(* CODESYS project tcl_baseclasses.library
   Company: Red Rock Controls Limited
   Description: Naming convention updated
   Version: 1.1.0.0
   Placeholder: tcl_BaseClasses
   Author: Roger Christopher
   Title: tcl_BaseClasses

Project tree, tasks and I/O mapping:
  libraries: Tc2_Standard, * (Beckhoff Automation GmbH); Tc2_System, * (Beckhoff Automation GmbH); Tc2_Utilities, * (Beckhoff Automation GmbH); Tc3_DynamicMemory, * (Beckhoff Automation GmbH); Tc3_EventLogger, * (Beckhoff Automation GmbH); Tc3_Module, * (Beckhoff Automation GmbH); tcl_StringUtils, * (Red Rock Controls Limited)
  Classes/
    Event Framework/
      Event Base Class/
        interface I_Event: AddEventHandler, Args, ClearEventHandlers, Raise
        function block T_EventBase [ST]: AddEventHandler, Args, CallHandler, ClearEventHandlers, IsHandlerSupported, Raise
      Event Handler Base/
        interface I_EventHandlerBase
      List Of Handlers/
        function block T_ListOfEventHandlers [ST]: AddHandler, Clear, Count, FB_exit, FB_init, GetHandler
    Execution/
      Execution/
        interface I_Execution: Abort, Clear, Start, Aborted, Busy, Done, Error, ErrorId, Event_OnAbort, Event_OnError, Notification_OnAbort, Notification_OnError, Ready, Starting
        function block T_Execution [ST]: Abort, Clear, FB_init, SetAborted, SetBusy, SetDone, SetError, Start, Aborted, Aborting, Busy, Done, Error, ErrorId, Event_OnAbort, Event_OnError, Notification_OnAbort, Notification_OnError, Ready, Starting, State
        data type T_ExecutionState
    Function Block Wrappers/
      Classes/
        function block T_Counter [ST]: Dec, Inc, Reset, Value, ValueAsTArg
        function block T_FallingEdge [ST]: EdgeDetected, Test
        function block T_OffTimer [ST]: Delay, FB_init, OutputState, PresetTime
        function block T_OnTimer [ST]: Delay, FB_init, OutputState, PresetTime, Reset, Run
        function block T_PulseTimer [ST]: FB_init, OutputState, PresetTime, Pulse, Reset, Run
        function block T_RisingEdge [ST]: EdgeDetected, Test
        function block T_StructureCrcMonitor [ST]: Changed, Reset, Test
        function block T_ValueMonitor [ST]: Changed, CurrentValue, PreviousValue, Reset, Test
        function block T_ValueMonitorEx [ST]: Changed, Reset, Test
      Event Logging/
        function F_LogError [ST]
        function F_LogMessage [ST]
        function F_LogWarning [ST]
    Notifications/
      Handler Interface/
        interface I_NotificationHandler: OnNotificationReceived
        function block T_NotificationHandler [ST]: IsRaised, NotificationArgs, OnNotificationReceived
      List Of Handlers/
        function block T_ListONotificationHandlers [ST]: AddHandler, Clear, Count, FB_exit, FB_init, GetHandler
      Notification Class/
        interface I_Notification: AddNotificationHandler, ClearNotificationHandlers, Raise, SetNotificationId, Args, Name, NotificationId
        function block T_Notification [ST]: AddNotificationHandler, ClearNotificationHandlers, FB_init, Raise, SetNotificationId, stripName, Args, Name, NotificationId
    Stream/
      interface I_StreamReader: Read_BLOB, Read_BOOL, Read_BYTE, Read_DINT, Read_INT, Read_LINT, Read_LREAL, Read_PVOID, Read_REAL, Read_STRING, Read_UDINT, Read_UINT, Read_ULINT, Seek, BufferAddress, ByteCount, Position, StreamLength
      interface I_StreamWriter: Add_BLOB, Add_BOOL, Add_BYTE, Add_DINT, Add_INT, Add_LINT, Add_LREAL, Add_PVOID, Add_REAL, Add_STRING, Add_UDINT, Add_UINT, Add_ULINT, Clear, Seek
      function block T_Stream [ST]: _ResizeIfNecessary, Add_BLOB, Add_BOOL, Add_BYTE, Add_DINT, Add_INT, Add_LINT, Add_LREAL, Add_PVOID, Add_REAL, Add_STRING, Add_UDINT, Add_UINT, Add_ULINT, Clear, CopyFromStreamReader, FB_exit, FB_init, Init, Read_BLOB, Read_BOOL, Read_BYTE, Read_DINT, Read_INT, Read_LINT, Read_LREAL, Read_PVOID, Read_REAL, Read_STRING, Read_UDINT, Read_UINT, Read_ULINT, Resize, Seek, BufferAddress, ByteCount, Position, StreamLength
  Events/
    Assertion Failed/
      interface I_EventHandler_OnAssertionFailed: OnAssertionFailed
      function block T_Event_AssertionFailed [ST]: CallHandler, IsHandlerSupported
    Execution Aborted/
      interface I_EventHandler_OnExecutionAborted: OnExecutionAborted
      function block T_Event_ExecutionAborted [ST]: CallHandler, IsHandlerSupported
    Execution Failed/
      interface I_EventHandler_OnExecutionFailed: OnExecutionFailed
      function block T_Event_ExecutionFailed [ST]: CallHandler, IsHandlerSupported
  Functions/
    function F_Assert [ST]
    function F_ClearMem [ST]
    function F_DINT_TO_UDINT [ST]
    function F_Equals [ST]
    function F_GetAdsPort [ST]
    function F_GetTaskTime [ST]
    function F_NotEqual [ST]
    function F_UDINT_TO_DINT [ST]
  GVLs/
    global variables GlobalEvents
    global variables GlobalVariables
*)

// Classes/Execution/Execution/T_ExecutionState
{attribute 'qualified_only'}
{attribute 'strict'}
TYPE T_ExecutionState :
(
    Ready := 0,
	Starting,
    Busy,
    Aborting);
END_TYPE

// GVLs/GlobalEvents
(*
Global event instances 
These events are raised by all instances of T_Execution by default when an error occurs
This behaviour can be overidden by setting the Event_OnError or Event_OnAbort properties
of the instance of T_Execution to 0
*)
{attribute 'qualified_only'}
VAR_GLOBAL
    Event_OnError           : T_Event_ExecutionFailed;
    Event_OnAbort           : T_Event_ExecutionAborted;
    Event_AssertionFailed   : T_Event_AssertionFailed;
    
    Notification_ExecutionFailed  : T_Notification;
    Notification_ExecutionAborted : T_Notification;
    Notification_AssertionFailed  : T_Notification;
    
END_VAR

// GVLs/GlobalVariables
{attribute 'qualified_only'}
VAR_GLOBAL
    //Message : FB_TcMessage;
END_VAR

// Classes/Event Framework/Event Base Class/I_Event
INTERFACE I_Event

METHOD AddEventHandler : I_Event
VAR_INPUT
    Handler : I_EventHandlerBase;
END_VAR
END_METHOD

PROPERTY Args : I_StreamWriter
GET
END_GET
END_PROPERTY

METHOD ClearEventHandlers : I_Event
VAR_INPUT
END_VAR
END_METHOD

METHOD Raise
END_METHOD

END_INTERFACE

// Classes/Event Framework/Event Handler Base/I_EventHandlerBase
INTERFACE I_EventHandlerBase EXTENDS __SYSTEM.IQueryInterface

END_INTERFACE

// Classes/Stream/I_StreamWriter
INTERFACE I_StreamWriter

METHOD Add_BLOB : I_StreamWriter
VAR_INPUT
    Value : ANY;
END_VAR
END_METHOD

METHOD Add_BOOL : I_StreamWriter
VAR_INPUT
    Value : BOOL;
END_VAR
END_METHOD

METHOD Add_BYTE : I_StreamWriter
VAR_INPUT
    Value : BYTE;
END_VAR
END_METHOD

METHOD Add_DINT : I_StreamWriter
VAR_INPUT
    Value : DINT;
END_VAR
END_METHOD

METHOD Add_INT : I_StreamWriter
VAR_INPUT
    Value : INT;
END_VAR
END_METHOD

METHOD Add_LINT : I_StreamWriter
VAR_INPUT
    Value : LINT;
END_VAR
END_METHOD

METHOD Add_LREAL : I_StreamWriter
VAR_INPUT
    Value : LREAL;
END_VAR
END_METHOD

METHOD Add_PVOID : I_StreamWriter
VAR_INPUT
    Value : PVOID;
END_VAR
END_METHOD

METHOD Add_REAL : I_StreamWriter
VAR_INPUT
    Value : REAL;
END_VAR
END_METHOD

METHOD Add_STRING : I_StreamWriter
VAR_INPUT
    Value : STRING(255);
END_VAR
END_METHOD

METHOD Add_UDINT : I_StreamWriter
VAR_INPUT
    Value : UDINT;
END_VAR
END_METHOD

METHOD Add_UINT : I_StreamWriter
VAR_INPUT
    Value : UINT;
END_VAR
END_METHOD

METHOD Add_ULINT : I_StreamWriter
VAR_INPUT
    Value : ULINT;
END_VAR
END_METHOD

METHOD Clear : I_StreamWriter
END_METHOD

METHOD Seek: I_StreamWriter
VAR_INPUT
    Position : UDINT;
END_VAR
END_METHOD

END_INTERFACE

// Classes/Event Framework/Event Base Class/T_EventBase
{attribute 'reflection'}
FUNCTION_BLOCK ABSTRACT T_EventBase IMPLEMENTS I_Event
VAR
    EventHandlers : T_ListOfEventHandlers(Capacity := 5);
    
    {attribute 'instance-path'} {attribute 'no_init'}
    EventName : T_MaxString; // Automatically initialised with the full name of the instance   
    
    EventArgs : T_Stream(StreamLength := 8);
    
    Message_EventHandlerNotImplemented : FB_TcMessage;
END_VAR

METHOD AddEventHandler : I_Event
VAR_INPUT
    Handler : I_EventHandlerBase;
END_VAR
IF IsHandlerSupported(Handler) THEN
    EventHandlers.AddHandler(Handler);
//ELSE
//    IF Message_EventHandlerNotImplemented.nEventId = 0 THEN
//        Message_EventHandlerNotImplemented.CreateEx(
//            stEventEntry := TC_EVENTS.tcl_BaseClassEvents.EventHandlerNotImplemented,
//            ipSourceInfo := 0);
//    END_IF
//    Message_EventHandlerNotImplemented.Send(0);

END_IF
AddEventHandler := THIS^;
END_METHOD

PROPERTY PUBLIC Args : I_StreamWriter
GET
Args := EventArgs;
END_GET
END_PROPERTY

METHOD ABSTRACT CallHandler
VAR_INPUT
    HandlerBase : I_EventHandlerBase;
    EventArgs : I_StreamReader;
END_VAR
END_METHOD

METHOD ClearEventHandlers : I_Event
EventHandlers.Clear();
ClearEventHandlers := THIS^;
END_METHOD

METHOD ABSTRACT IsHandlerSupported : BOOL
VAR_INPUT
    HandlerBase : I_EventHandlerBase;
END_VAR
END_METHOD

METHOD Raise
VAR
    HandlerBase : I_EventHandlerBase;
    i : UDINT;
END_VAR
IF EventHandlers.Count > 0 THEN
    FOR i := 0 TO EventHandlers.Count - 1 DO
        HandlerBase := EventHandlers.GetHandler(i);
        IF HandlerBase <> 0 THEN
            EventArgs.Seek(0); // to ensure that each handler reads args from start of the stream
            CallHandler(HandlerBase,EventArgs);
        END_IF
    END_FOR
END_IF
EventArgs.Clear(); // to leave event args empty for next time event is raised
END_METHOD

END_FUNCTION_BLOCK

// Classes/Event Framework/List Of Handlers/T_ListOfEventHandlers
{attribute 'hide'}
FUNCTION_BLOCK T_ListOfEventHandlers
VAR
    Buffer : FB_DynMem_Buffer(ipMemMan:= DynamicMemoryManager);
    DynamicMemoryManager : FB_DynMem_Manager;

    pHandler : POINTER TO I_EventHandlerBase;
    HandlerCount : UDINT;
    Capacity : UDINT;
END_VAR

METHOD AddHandler
VAR_INPUT
    Handler : I_EventHandlerBase;
END_VAR
IF Count = Capacity THEN
    Capacity := Capacity * 2;
    Buffer.Resize(
        nSize     := Capacity * SIZEOF(PVOID),
        bPreserve := TRUE,
        bReset    := FALSE);
    pHandler := Buffer.pBuffer;
END_IF

pHandler[HandlerCount] := Handler;
HandlerCount := HandlerCount + 1;
END_METHOD

METHOD Clear
VAR_INPUT
END_VAR
Buffer.Clear();
HandlerCount := 0;
END_METHOD

PROPERTY Count : UDINT
GET
Count := HandlerCount;
END_GET
END_PROPERTY

METHOD FB_exit : BOOL
VAR_INPUT
	bInCopyCode : BOOL; // if TRUE, the exit method is called for exiting an instance that is copied afterwards (online change).
END_VAR
IF NOT bInCopyCode THEN
    Buffer.DeleteBuffer();
    pHandler := 0;
END_IF
END_METHOD

METHOD FB_init : BOOL
VAR_INPUT
	bInitRetains : BOOL; // if TRUE, the retain variables are initialized (warm start / cold start)
	bInCopyCode : BOOL;  // if TRUE, the instance afterwards gets moved into the copy code (online change)
    Capacity : UDINT;
END_VAR
Buffer.CreateBuffer(
    nSize := Capacity * SIZEOF(PVOID),
    bReset := TRUE);
    
pHandler := Buffer.pBuffer;
THIS^.Capacity := Capacity;
END_METHOD

METHOD GetHandler : I_EventHandlerBase
VAR_INPUT
    Index : UDINT;
END_VAR
IF Index < HandlerCount AND Index >= 0 THEN 
    GetHandler := pHandler[Index];
END_IF
END_METHOD

END_FUNCTION_BLOCK

// Classes/Stream/T_Stream
FUNCTION_BLOCK T_Stream IMPLEMENTS I_StreamWriter, I_StreamReader
VAR
    
    MemoryManager : FB_DynMem_Manager;
    Buffer : FB_DynMem_Buffer(ipMemMan:= MemoryManager);
    pBuffer : POINTER TO BYTE;
    
    _StreamLength : UDINT := 4;
    _Position : UDINT;
    _ByteCount : UDINT;
END_VAR

METHOD PRIVATE _ResizeIfNecessary
VAR_INPUT
    SpaceRequired : UDINT;
END_VAR
IF _Position + SpaceRequired > _StreamLength THEN
    Resize(StreamLength := _Position + SpaceRequired);
END_IF
END_METHOD

METHOD Add_BLOB : I_StreamWriter
VAR_INPUT
    Value : ANY;
END_VAR
VAR
    pValue : POINTER TO BYTE;
END_VAR
_ResizeIfNecessary(SpaceRequired := DINT_TO_UDINT(Value.diSize));

MEMCPY(
    destAddr:= pBuffer + _Position, 
    srcAddr := Value.pValue, 
    n       := DINT_TO_UDINT(Value.diSize));

_Position  := _Position + DINT_TO_UDINT(Value.diSize); 
_ByteCount := _ByteCount + DINT_TO_UDINT(Value.diSize); 
   
Add_BLOB := THIS^;
END_METHOD

METHOD Add_BOOL : I_StreamWriter
VAR_INPUT
    Value : BOOL;
END_VAR
VAR
    pValue : POINTER TO BOOL;
END_VAR
_ResizeIfNecessary(SpaceRequired := SIZEOF(Value));

pValue := pBuffer + _Position;
pValue^ := Value;
_Position := _Position + SIZEOF(Value); 
_ByteCount := _ByteCount + SIZEOF(Value); 
   
Add_BOOL := THIS^;
END_METHOD

METHOD Add_BYTE : I_StreamWriter
VAR_INPUT
    Value : BYTE;
END_VAR
VAR
    pValue : POINTER TO BYTE;
END_VAR
_ResizeIfNecessary(SpaceRequired := SIZEOF(Value));

pValue := pBuffer + _Position;
pValue^ := Value;
_Position := _Position + SIZEOF(Value); 
_ByteCount := _ByteCount + SIZEOF(Value); 

Add_BYTE := THIS^;
END_METHOD

METHOD Add_DINT : I_StreamWriter
VAR_INPUT
    Value : DINT;
END_VAR
VAR
    pValue : POINTER TO DINT;
END_VAR
_ResizeIfNecessary(SpaceRequired := SIZEOF(Value));

pValue := pBuffer + _Position;
pValue^ := Value;
_Position := _Position + SIZEOF(Value); 
_ByteCount := _ByteCount + SIZEOF(Value); 

   
Add_DINT := THIS^;
END_METHOD

METHOD Add_INT : I_StreamWriter
VAR_INPUT
    Value : INT;
END_VAR
VAR
    pValue : POINTER TO INT;
END_VAR
_ResizeIfNecessary(SpaceRequired := SIZEOF(Value));

pValue := pBuffer + _Position;
pValue^ := Value;
_Position := _Position + SIZEOF(Value);    
_ByteCount := _ByteCount + SIZEOF(Value); 


Add_INT := THIS^;
END_METHOD

METHOD Add_LINT : I_StreamWriter
VAR_INPUT
    Value : LINT;
END_VAR
VAR
    pValue : POINTER TO LINT;
END_VAR
_ResizeIfNecessary(SpaceRequired := SIZEOF(Value));

pValue := pBuffer + _Position;
pValue^ := Value;
_Position := _Position + SIZEOF(Value); 
_ByteCount := _ByteCount + SIZEOF(Value); 

   
Add_LINT := THIS^;
END_METHOD

METHOD Add_LREAL : I_StreamWriter
VAR_INPUT
    Value : LREAL;
END_VAR
VAR
    pValue : POINTER TO LREAL;
END_VAR
_ResizeIfNecessary(SpaceRequired := SIZEOF(Value));

pValue := pBuffer + _Position;
pValue^ := Value;
_Position := _Position + SIZEOF(Value);    
_ByteCount := _ByteCount + SIZEOF(Value); 


Add_LREAL := THIS^;
END_METHOD

METHOD Add_PVOID : I_StreamWriter
VAR_INPUT
    Value : PVOID;
END_VAR
VAR
    pValue : POINTER TO PVOID;
END_VAR
_ResizeIfNecessary(SpaceRequired := SIZEOF(Value));

pValue := pBuffer + _Position;
pValue^ := Value;
_Position := _Position + SIZEOF(Value); 
_ByteCount := _ByteCount + SIZEOF(Value); 

   
Add_PVOID := THIS^;
END_METHOD

METHOD Add_REAL : I_StreamWriter
VAR_INPUT
    Value : REAL;
END_VAR
VAR
    pValue : POINTER TO REAL;
END_VAR
_ResizeIfNecessary(SpaceRequired := SIZEOF(Value));

pValue := pBuffer + _Position;
pValue^ := Value;
_Position := _Position + SIZEOF(Value);    
_ByteCount := _ByteCount + SIZEOF(Value); 


Add_REAL := THIS^;
END_METHOD

METHOD Add_STRING : I_StreamWriter // adds any string length as we only store the chars + null byte
VAR_INPUT
    Value : STRING(255);
END_VAR
VAR
    StringSize : UDINT; // number of characters plus the null termination byte
END_VAR
StringSize := INT_TO_UDINT(LEN(Value) + 1);

_ResizeIfNecessary(SpaceRequired := StringSize);  // only storing the characters and the null termination byte

MEMCPY(
    destAddr := pBuffer + _Position,
    srcAddr  := ADR(Value),
    n        := StringSize);


_Position := _Position + StringSize;    
_ByteCount := _ByteCount + StringSize; 


Add_STRING := THIS^;
END_METHOD

METHOD Add_UDINT : I_StreamWriter
VAR_INPUT
    Value : UDINT;
END_VAR
VAR
    pValue : POINTER TO UDINT;
END_VAR
_ResizeIfNecessary(SpaceRequired := SIZEOF(Value));

pValue := pBuffer + _Position;
pValue^ := Value;
_Position := _Position + SIZEOF(Value);    
_ByteCount := _ByteCount + SIZEOF(Value); 


Add_UDINT := THIS^;
END_METHOD

METHOD Add_UINT : I_StreamWriter
VAR_INPUT
    Value : UINT;
END_VAR
VAR
    pValue : POINTER TO UINT;
END_VAR
_ResizeIfNecessary(SpaceRequired := SIZEOF(Value));

pValue := pBuffer + _Position;
pValue^ := Value;
_Position := _Position + SIZEOF(Value);    
_ByteCount := _ByteCount + SIZEOF(Value); 


Add_UINT := THIS^;
END_METHOD

METHOD Add_ULINT : I_StreamWriter
VAR_INPUT
    Value : ULINT;
END_VAR
VAR
    pValue : POINTER TO ULINT;
END_VAR
_ResizeIfNecessary(SpaceRequired := SIZEOF(Value));

pValue := pBuffer + _Position;
pValue^ := Value;
_Position := _Position + SIZEOF(Value); 
_ByteCount := _ByteCount + SIZEOF(Value); 

   
Add_ULINT := THIS^;
END_METHOD

METHOD Clear : I_StreamWriter
Buffer.Clear();
_Position := 0;
_ByteCount := 0;
pBuffer := Buffer.pBuffer;
Clear := THIS^;
END_METHOD

METHOD CopyFromStreamReader
VAR_INPUT
    StreamToCopyFrom : I_StreamReader;
END_VAR
IF StreamToCopyFrom.StreamLength > THIS^.StreamLength THEN
    Resize(StreamToCopyFrom.StreamLength);
END_IF

MEMCPY(
    destAddr := Buffer.pBuffer,
    srcAddr  := StreamToCopyFrom.BufferAddress,
    n        := StreamToCopyFrom.StreamLength);
    
THIS^._ByteCount    := StreamToCopyFrom.ByteCount;
THIS^._StreamLength := StreamToCopyFrom.StreamLength;
THIS^._Position     := 0;
END_METHOD

METHOD FB_exit : BOOL
VAR_INPUT
	bInCopyCode : BOOL; // if TRUE, the exit method is called for exiting an instance that is copied afterwards (online change).
END_VAR
IF NOT bInCopyCode THEN
    Buffer.DeleteBuffer();
END_IF
END_METHOD

METHOD FB_init : BOOL
VAR_INPUT
	bInitRetains : BOOL; // if TRUE, the retain variables are initialized (warm start / cold start)
	bInCopyCode : BOOL;  // if TRUE, the instance afterwards gets moved into the copy code (online change)
    StreamLength : UDINT;
END_VAR
IF NOT bInCopyCode THEN
    Init(StreamLength);
END_IF
END_METHOD

METHOD Init
VAR_INPUT
    StreamLength : UDINT;
END_VAR
IF Buffer.bAvailable THEN
    Buffer.DeleteBuffer();
END_IF

_StreamLength := StreamLength;
Buffer.CreateBuffer(nSize := _StreamLength, bReset := TRUE);
_Position := 0;
_ByteCount := 0;
pBuffer := Buffer.pBuffer;
END_METHOD

METHOD Read_BLOB
VAR_INPUT
    Value : ANY;
END_VAR

VAR
    pValue : POINTER TO BYTE;
    Result : BYTE;
END_VAR
IF _Position + DINT_TO_UDINT(Value.diSize) <= _StreamLength THEN
    
MEMCPY(
    destAddr:= Value.pValue, 
    srcAddr := pBuffer + _Position, 
    n       := DINT_TO_UDINT(Value.diSize));

    _Position := _Position + DINT_TO_UDINT(Value.diSize);   
END_IF
END_METHOD

METHOD Read_BOOL : BOOL;
VAR
    pValue : POINTER TO BOOL;
    Result : BOOL;
END_VAR
IF _Position + SIZEOF(Result) <= _StreamLength THEN
    pValue := pBuffer + _Position;
    Result := pValue^;
    _Position := _Position + SIZEOF(Result);   
    Read_BOOL := Result; 
END_IF
END_METHOD

METHOD Read_BYTE : BYTE;
VAR
    pValue : POINTER TO BYTE;
    Result : BYTE;
END_VAR
IF _Position + SIZEOF(Result) <= _StreamLength THEN
    pValue := pBuffer + _Position;
    Result := pValue^;
    _Position := _Position + SIZEOF(Result);   
    Read_BYTE := Result; 
END_IF
END_METHOD

METHOD Read_DINT : DINT;
VAR
    pValue : POINTER TO DINT;
    Result : DINT;
END_VAR
IF _Position + SIZEOF(Result) <= _StreamLength THEN
    pValue := pBuffer + _Position;
    Result := pValue^;
    _Position := _Position + SIZEOF(Result);   
    Read_DINT := Result; 
END_IF
END_METHOD

METHOD Read_INT : INT;
VAR
    pValue : POINTER TO INT;
    Result : INT;
END_VAR
IF _Position + SIZEOF(Result) <= _StreamLength THEN
    pValue := pBuffer + _Position;
    Result := pValue^;
    _Position := _Position + SIZEOF(Result);   
    Read_INT := Result; 
END_IF
END_METHOD

METHOD Read_LINT : LINT;
VAR
    pValue : POINTER TO LINT;
    Result : LINT;
END_VAR
IF _Position + SIZEOF(Result) <= _StreamLength THEN
    pValue := pBuffer + _Position;
    Result := pValue^;
    _Position := _Position + SIZEOF(Result);   
    Read_LINT := Result; 
END_IF
END_METHOD

METHOD Read_LREAL : LREAL;
VAR
    pValue : POINTER TO LREAL;
    Result : LREAL;
END_VAR
IF _Position + SIZEOF(Result) <= _StreamLength THEN
    pValue := pBuffer + _Position;
    Result := pValue^;
    _Position := _Position + SIZEOF(Result);   
    Read_LREAL := Result; 
END_IF
END_METHOD

METHOD Read_PVOID : PVOID;
VAR
    pValue : POINTER TO PVOID;
    Result : PVOID;
END_VAR
IF _Position + SIZEOF(Result) <= _StreamLength THEN
    pValue := pBuffer + _Position;
    Result := pValue^;
    _Position := _Position + SIZEOF(Result);   
    Read_PVOID := Result; 
END_IF
END_METHOD

METHOD Read_REAL : REAL;
VAR
    pValue : POINTER TO REAL;
    Result : REAL;
END_VAR
IF _Position + SIZEOF(Result) <= _StreamLength THEN
    pValue := pBuffer + _Position;
    Result := pValue^;
    _Position := _Position + SIZEOF(Result);   
    Read_REAL := Result; 
END_IF
END_METHOD

METHOD Read_STRING : STRING(255);
VAR
    pValue : POINTER TO STRING(255);
    StringSize : UDINT; // number of characters plus the null termination byte
END_VAR
pValue := pBuffer + _Position;

StringSize := INT_TO_UDINT(LEN(pValue^) + 1);

IF _Position + StringSize <= _StreamLength THEN // end of string is in the buffer, so proceed...
    _Position := _Position + StringSize;   
    Read_STRING := pValue^;
END_IF
END_METHOD

METHOD Read_UDINT : UDINT;
VAR
    pValue : POINTER TO UDINT;
    Result : UDINT;
END_VAR
IF _Position + SIZEOF(Result) <= _StreamLength THEN
    pValue := pBuffer + _Position;
    Result := pValue^;
    _Position := _Position + SIZEOF(Result);   
    Read_UDINT := Result; 
END_IF
END_METHOD

METHOD Read_UINT : UINT;
VAR
    pValue : POINTER TO UINT;
    Result : UINT;
END_VAR
IF _Position + SIZEOF(Result) <= _StreamLength THEN
    pValue := pBuffer + _Position;
    Result := pValue^;
    _Position := _Position + SIZEOF(Result);   
    Read_UINT := Result; 
END_IF
END_METHOD

METHOD Read_ULINT : ULINT;
VAR
    pValue : POINTER TO ULINT;
    Result : ULINT;
END_VAR
IF _Position + SIZEOF(Result) <= _StreamLength THEN
    pValue := pBuffer + _Position;
    Result := pValue^;
    _Position := _Position + SIZEOF(Result);   
    Read_ULINT := Result; 
END_IF
END_METHOD

METHOD Resize
VAR_INPUT
    StreamLength : UDINT;
END_VAR
Buffer.Resize(nSize := StreamLength, bPreserve := TRUE, bReset := FALSE);
_StreamLength := StreamLength;
pBuffer := Buffer.pBuffer;
END_METHOD

METHOD Seek : I_StreamWriter
VAR_INPUT
    Position : UDINT;
END_VAR
IF Position <= _StreamLength THEN
    THIS^._Position := Position;
END_IF
Seek := THIS^;
END_METHOD

PROPERTY BufferAddress : PVOID
GET
BufferAddress := Buffer.pBuffer;
END_GET
END_PROPERTY

PROPERTY ByteCount : UDINT
GET
ByteCount := _ByteCount;
END_GET
END_PROPERTY

PROPERTY Position : UDINT
GET
Position := _Position;
END_GET
END_PROPERTY

PROPERTY StreamLength : UDINT
GET
StreamLength := _StreamLength;
END_GET
END_PROPERTY

END_FUNCTION_BLOCK

// Classes/Stream/I_StreamReader
INTERFACE I_StreamReader

METHOD Read_BLOB
VAR_INPUT
    Value : ANY;
END_VAR
END_METHOD

METHOD Read_BOOL : BOOL;
END_METHOD

METHOD Read_BYTE : BYTE;
END_METHOD

METHOD Read_DINT : DINT;
END_METHOD

METHOD Read_INT : INT;
END_METHOD

METHOD Read_LINT : LINT;
END_METHOD

METHOD Read_LREAL : LREAL;
END_METHOD

METHOD Read_PVOID : PVOID;
END_METHOD

METHOD Read_REAL : REAL;
END_METHOD

METHOD Read_STRING : STRING(255);
END_METHOD

METHOD Read_UDINT : UDINT;
END_METHOD

METHOD Read_UINT : UINT;
END_METHOD

METHOD Read_ULINT : ULINT;
END_METHOD

METHOD Seek: I_StreamWriter
VAR_INPUT
    Position : UDINT;
END_VAR
END_METHOD

PROPERTY BufferAddress : PVOID
GET
END_GET
END_PROPERTY

PROPERTY ByteCount : UDINT
GET
END_GET
END_PROPERTY

PROPERTY Position : UDINT
GET
END_GET
END_PROPERTY

PROPERTY StreamLength : UDINT
GET
END_GET
END_PROPERTY

END_INTERFACE

// Classes/Execution/Execution/I_Execution
INTERFACE I_Execution

METHOD Abort 
VAR_INPUT
END_VAR
END_METHOD

METHOD Clear 
VAR_INPUT
END_VAR
END_METHOD

METHOD Start : BOOL // returns TRUE if start request accepted (i.e State was Ready)
VAR_INPUT
END_VAR
END_METHOD

PROPERTY Aborted : BOOL
GET
END_GET
END_PROPERTY

PROPERTY Busy : BOOL
GET
END_GET
END_PROPERTY

PROPERTY Done : BOOL
GET
END_GET
END_PROPERTY

PROPERTY Error : BOOL
GET
END_GET
END_PROPERTY

PROPERTY ErrorId : UDINT
GET
END_GET
END_PROPERTY

PROPERTY Event_OnAbort : I_Event
GET
END_GET
SET
END_SET
END_PROPERTY

PROPERTY Event_OnError : I_Event
GET
END_GET
SET
END_SET
END_PROPERTY

PROPERTY Notification_OnAbort : I_Notification
GET
END_GET
SET
END_SET
END_PROPERTY

PROPERTY Notification_OnError : I_Notification
GET
END_GET
SET
END_SET
END_PROPERTY

PROPERTY Ready : BOOL
GET
END_GET
END_PROPERTY

PROPERTY Starting : BOOL
GET
END_GET
END_PROPERTY

END_INTERFACE

// Classes/Notifications/Notification Class/I_Notification
INTERFACE I_Notification

METHOD AddNotificationHandler : I_Notification
VAR_INPUT
    Handler : I_NotificationHandler;
END_VAR
END_METHOD

METHOD ClearNotificationHandlers : I_Notification
VAR_INPUT
END_VAR
END_METHOD

METHOD Raise
END_METHOD

METHOD SetNotificationId : I_Notification
VAR_INPUT
    NotificationId : UDINT;
END_VAR
END_METHOD

PROPERTY Args : I_StreamWriter
GET
END_GET
END_PROPERTY

PROPERTY Name : T_MaxString
GET
END_GET
END_PROPERTY

PROPERTY NotificationId : UDINT
GET
END_GET
SET
END_SET
END_PROPERTY

END_INTERFACE

// Classes/Notifications/Handler Interface/I_NotificationHandler
INTERFACE I_NotificationHandler EXTENDS __SYSTEM.IQueryInterface

METHOD OnNotificationReceived
VAR_INPUT
    NotificationId   : UDINT;
    NotificationName : T_MaxString;
    Args             : I_StreamReader;
END_VAR
END_METHOD

END_INTERFACE

// Classes/Execution/Execution/T_Execution
(*
:Class for handling communications between a client requesting a service 
:and a server providing the service
*)
{attribute 'reflection'}
FUNCTION_BLOCK T_Execution IMPLEMENTS I_Execution
VAR
    _State      : T_ExecutionState;
    _Done       : BOOL;
    _Error      : BOOL;
    _Aborted    : BOOL;
    
    {attribute 'displaymode':='hex'}
    _ErrorId    : UDINT;
    
    {attribute 'instance-path'} {attribute 'no_init'}
    Name        : T_MaxString; // Automatically initialised with the full name of the instance
    
    _Event_OnError : I_Event;
    _Event_OnAbort : I_Event;
    
    _Notification_OnError : I_Notification;
    _Notification_OnAbort : I_Notification;
    
    SourceInfo : FB_TcSourceInfo;
    
    Message_ExecutionError : FB_TcMessage;
    Message_ExecutionAborted : FB_TcMessage;
    Message_ExecutionNotReady : FB_TcMessage;
END_VAR

// Requests that the current operation be aborted - set the State to Aborting
METHOD Abort
// Aborting must be handled by parent class - cleanup and set Ready state
_State := T_ExecutionState.Aborting;
END_METHOD

// Clears the results flags provided State = Ready
METHOD Clear
IF _State = T_ExecutionState.Ready  THEN
    _Done    := FALSE;
    _Aborted := FALSE;
    _Error   := FALSE;
    _ErrorId := 0;
    
ELSE
    IF _Event_OnError <> 0 THEN
        _Event_OnError.Args.Add_STRING(F_FormatString1(
                                        Format := 'Clear requested while not ready in %s',
                                        Arg1   := F_STRING(Name)));
        _Event_OnError.Raise();
    END_IF
END_IF
END_METHOD

// Individual T_Execution events are assigned here to the global events 
// so by default, all errors/aborts raise these global events
// This can be overidden for individual instances or T_Execution 
// by setting the Event properties to zero (or another event)
METHOD FB_init : BOOL
VAR_INPUT
	bInitRetains : BOOL; // if TRUE, the retain variables are initialized (warm start / cold start)
	bInCopyCode : BOOL;  // if TRUE, the instance afterwards gets moved into the copy code (online change)
END_VAR
_Event_OnAbort := GlobalEvents.Event_OnAbort;
_Event_OnError := GlobalEvents.Event_OnError;
_Notification_OnAbort := GlobalEvents.Notification_ExecutionAborted;
_Notification_OnError := GlobalEvents.Notification_ExecutionFailed;

SourceInfo.sName := Name;
END_METHOD

METHOD SetAborted // used when implementing class signals Aborted
VAR
    EventData : T_MaxString;
END_VAR
IF _State = T_ExecutionState.Starting OR _State = T_ExecutionState.Busy THEN
    _Aborted := TRUE;
    _State := T_ExecutionState.Ready;
    
    IF _Event_OnAbort <> 0 THEN
        _Event_OnAbort.Args.Add_STRING(F_FormatString1('Execution aborted in %s',F_STRING(Name)));
        _Event_OnAbort.Raise();
    END_IF  

    IF _Notification_OnAbort <> 0 THEN
        _Notification_OnAbort.Args.Add_STRING(F_FormatString1('Execution aborted in %s',F_STRING(Name)));
        _Notification_OnAbort.Raise();
    END_IF  

//    IF Message_ExecutionAborted.nEventId = 0 THEN
//        Message_ExecutionAborted.CreateEx(
//            stEventEntry := TC_EVENTS.tcl_BaseClassEvents.ExecutionAborted,
//            ipSourceInfo := 0);
//    END_IF
//    Message_ExecutionAborted.Send(0);
END_IF

IF _State = T_ExecutionState.Aborting THEN
    _Aborted := TRUE;
    _State := T_ExecutionState.Ready;
END_IF
END_METHOD

METHOD SetBusy
VAR_INPUT
END_VAR
IF _State = T_ExecutionState.Starting THEN
    _State := T_ExecutionState.Busy;
END_IF
END_METHOD

METHOD SetDone
VAR_INPUT
END_VAR
IF _State = T_ExecutionState.Starting OR _State = T_ExecutionState.Busy THEN
    _Done := TRUE;
    _State := T_ExecutionState.Ready;
END_IF
END_METHOD

METHOD SetError
VAR_INPUT
    ErrorId : UDINT;
END_VAR
IF _State = T_ExecutionState.Starting OR _State = T_ExecutionState.Busy THEN
    _Error   := TRUE;
    _ErrorId := ErrorId;
    _State   := T_ExecutionState.Ready;
    
    IF _Event_OnError <> 0 THEN
        _Event_OnError.Args.Add_STRING(F_FormatString2('Error 0x%0.4X in %s',F_UDINT(_ErrorId),F_STRING(Name)));
        _Event_OnError.Raise();
    END_IF
    
    IF _Notification_OnError <> 0 THEN
        _Notification_OnError.Args.Add_STRING(F_FormatString2('Error 0x%0.4X in %s',F_UDINT(_ErrorId),F_STRING(Name)));
        _Notification_OnError.Raise();
    END_IF
    
//    IF Message_ExecutionError.nEventId = 0 THEN
//        Message_ExecutionError.CreateEx(
//            stEventEntry := TC_EVENTS.tcl_BaseClassEvents.ExecutionError,
//            ipSourceInfo := 0);
//	END_IF
//    Message_ExecutionError.ipArguments.Clear().AddUDInt(_ErrorId);
//    Message_ExecutionError.Send(0);
END_IF
END_METHOD

METHOD Start : BOOL
VAR_INPUT
END_VAR
IF _State = T_ExecutionState.Ready  THEN
    _Done    := FALSE;
    _Aborted := FALSE;
    _Error   := FALSE;
    _ErrorId := 0;
    
    _State   := T_ExecutionState.Starting;
    Start    := TRUE; // Accepted
ELSE
    IF _Event_OnError <> 0 THEN
        _Event_OnError.Args.Add_STRING(F_FormatString1(
                                        Format := 'Start requested while not ready in %s',
                                        Arg1   := F_STRING(Name)));
        _Event_OnError.Raise();
    END_IF
    
//    IF Message_ExecutionNotReady.nEventId = 0 THEN
//        Message_ExecutionNotReady.CreateEx(
//            stEventEntry := TC_EVENTS.tcl_BaseClassEvents.ExecutionNotReady,
//            ipSourceInfo := 0);
//    END_IF
//    Message_ExecutionNotReady.Send(0);
    
END_IF
END_METHOD

PROPERTY Aborted : BOOL
GET
Aborted := _Aborted;
END_GET
END_PROPERTY

PROPERTY Aborting : BOOL
GET
Aborting := _State = T_ExecutionState.Aborting;
END_GET
END_PROPERTY

PROPERTY Busy : BOOL
GET
Busy := _State = T_ExecutionState.Busy;
END_GET
END_PROPERTY

PROPERTY Done : BOOL
GET
Done := _Done;
END_GET
END_PROPERTY

PROPERTY Error : BOOL
GET
Error := _Error;
END_GET
END_PROPERTY

PROPERTY ErrorId : UDINT
GET
ErrorId := _ErrorId;
END_GET
SET
_ErrorId := ErrorId;
END_SET
END_PROPERTY

PROPERTY Event_OnAbort : I_Event
GET
Event_OnAbort := _Event_OnAbort;
END_GET
SET
_Event_OnAbort := Event_OnAbort;
END_SET
END_PROPERTY

PROPERTY Event_OnError : I_Event
GET
Event_OnError := _Event_OnError;
END_GET
SET
_Event_OnError := Event_OnError;
END_SET
END_PROPERTY

PROPERTY Notification_OnAbort : I_Notification
GET
Notification_OnAbort := _Notification_OnAbort;
END_GET
SET
_Notification_OnAbort := Notification_OnAbort;
END_SET
END_PROPERTY

PROPERTY Notification_OnError : I_Notification
GET
Notification_OnError := _Notification_OnError;
END_GET
SET
_Notification_OnError := Notification_OnError;
END_SET
END_PROPERTY

PROPERTY Ready : BOOL
GET
Ready := _State = T_ExecutionState.Ready;
END_GET
END_PROPERTY

PROPERTY Starting : BOOL
GET
Starting := _State = T_ExecutionState.Starting;
END_GET
END_PROPERTY

PROPERTY State : T_ExecutionState
GET
State := _State;
END_GET
END_PROPERTY

END_FUNCTION_BLOCK

// Classes/Function Block Wrappers/Classes/T_Counter
FUNCTION_BLOCK T_Counter
VAR
    Count : DINT;
END_VAR

METHOD Dec : DINT
VAR_INPUT
END_VAR
Count := Count - 1;
Dec := Count;
END_METHOD

METHOD Inc : DINT
VAR_INPUT
END_VAR
Count := Count + 1;
Inc := Count;
END_METHOD

METHOD Reset
VAR_INPUT
END_VAR
Count := 0;
END_METHOD

PROPERTY Value : DINT
GET
Value := Count;
END_GET
SET
Count := Value;
END_SET
END_PROPERTY

PROPERTY ValueAsTArg : T_Arg
GET
ValueAsTArg := F_DINT(Count);
END_GET
END_PROPERTY

END_FUNCTION_BLOCK

// Classes/Function Block Wrappers/Classes/T_FallingEdge
FUNCTION_BLOCK T_FallingEdge
VAR
    F_TRIG1 : F_TRIG;
END_VAR

PROPERTY EdgeDetected : BOOL
GET
EdgeDetected := F_TRIG1.Q;
END_GET
END_PROPERTY

METHOD Test : BOOL
VAR_INPUT
    Value : BOOL;
END_VAR
F_TRIG1(CLK := Value);
Test := F_TRIG1.Q;
END_METHOD

END_FUNCTION_BLOCK

// Classes/Function Block Wrappers/Classes/T_OffTimer
FUNCTION_BLOCK T_OffTimer
VAR
    TOF1 : TOF;
END_VAR

METHOD Delay : BOOL
VAR_INPUT
    In : BOOL;
END_VAR
TOF1(IN := In);
Delay := TOF1.Q;
END_METHOD

METHOD FB_init : BOOL
VAR_INPUT
	bInitRetains : BOOL; // if TRUE, the retain variables are initialized (warm start / cold start)
	bInCopyCode : BOOL;  // if TRUE, the instance afterwards gets moved into the copy code (online change)
    PresetTime : LREAL; // seconds
END_VAR
TOF1.PT := LREAL_TO_TIME(PresetTime * 1000);
END_METHOD

PROPERTY OutputState : BOOL
GET
OutputState := TOF1.Q;
END_GET
END_PROPERTY

PROPERTY PresetTime : LREAL
GET
PresetTime := TIME_TO_LREAL(TOF1.PT)/1000.0; // in seconds
END_GET
SET
TOF1.PT := LREAL_TO_TIME(PresetTime * 1000);
END_SET
END_PROPERTY

END_FUNCTION_BLOCK

// Classes/Function Block Wrappers/Classes/T_OnTimer
FUNCTION_BLOCK T_OnTimer
VAR
    TON1 : TON;
END_VAR

METHOD Delay : BOOL
VAR_INPUT
    In : BOOL;
END_VAR
TON1(IN := In);
Delay := TON1.Q;
END_METHOD

METHOD FB_init : BOOL
VAR_INPUT
	bInitRetains : BOOL; // if TRUE, the retain variables are initialized (warm start / cold start)
	bInCopyCode : BOOL;  // if TRUE, the instance afterwards gets moved into the copy code (online change)
    PresetTime : LREAL; // seconds
END_VAR
TON1.PT := LREAL_TO_TIME(PresetTime * 1000);
END_METHOD

PROPERTY OutputState : BOOL
GET
OutputState := TON1.Q;
END_GET
END_PROPERTY

PROPERTY PresetTime : LREAL
GET
PresetTime := TIME_TO_LREAL(TON1.PT)/1000.0; // in seconds
END_GET
SET
TON1.PT := LREAL_TO_TIME(PresetTime * 1000);
END_SET
END_PROPERTY

METHOD Reset
TON1(IN := FALSE);
END_METHOD

METHOD Run : BOOL
TON1(IN := TRUE);
Run := TON1.Q;
END_METHOD

END_FUNCTION_BLOCK

// Classes/Function Block Wrappers/Classes/T_PulseTimer
FUNCTION_BLOCK T_PulseTimer
VAR
    TP1 : TP;
END_VAR

METHOD FB_init : BOOL
VAR_INPUT
	bInitRetains : BOOL; // if TRUE, the retain variables are initialized (warm start / cold start)
	bInCopyCode : BOOL;  // if TRUE, the instance afterwards gets moved into the copy code (online change)
    PresetTime : LREAL; // seconds
END_VAR
TP1.PT := LREAL_TO_TIME(PresetTime * 1000);
END_METHOD

PROPERTY OutputState : BOOL
GET
OutputState := TP1.Q;
END_GET
END_PROPERTY

PROPERTY PresetTime : LREAL
GET
PresetTime := TIME_TO_LREAL(TP1.PT)/1000.0; // in seconds
END_GET
SET
TP1.PT := LREAL_TO_TIME(PresetTime * 1000);
END_SET
END_PROPERTY

METHOD Pulse : BOOL
VAR_INPUT
    In : BOOL;
END_VAR
TP1(IN := In);
Pulse := TP1.Q;
END_METHOD

METHOD Reset
TP1(IN := FALSE);
END_METHOD

METHOD Run : BOOL
TP1(IN := TRUE);
Run := TP1.Q;
END_METHOD

END_FUNCTION_BLOCK

// Classes/Function Block Wrappers/Classes/T_RisingEdge
FUNCTION_BLOCK T_RisingEdge
VAR
    R_TRIG1 : R_TRIG;
END_VAR

PROPERTY EdgeDetected : BOOL
GET
EdgeDetected := R_TRIG1.Q;
END_GET
END_PROPERTY

METHOD Test : BOOL
VAR_INPUT
    Value : BOOL;
END_VAR
R_TRIG1(CLK := Value);
Test := R_TRIG1.Q;
END_METHOD

END_FUNCTION_BLOCK

// Classes/Function Block Wrappers/Classes/T_StructureCrcMonitor
{attribute 'no_explicit_call':= 'do not call this POU directly'}
FUNCTION_BLOCK T_StructureCrcMonitor
VAR
    _Changed : BOOL;
    Stored_CRC : WORD := 16#FFFF;
END_VAR

PROPERTY Changed : BOOL
GET
Changed := _Changed;
END_GET
END_PROPERTY

METHOD Reset
VAR_INPUT
END_VAR
Stored_CRC := 16#FFFF;
END_METHOD

METHOD Test
VAR_INPUT
    Structure : ANY;
END_VAR
VAR
    CRC : WORD;
END_VAR
CRC := F_DATA_TO_CRC16_CCITT(
            pData  := Structure.pValue, 
            cbData := DINT_TO_UDINT(Structure.diSize), 
            crc    := 0);

_Changed := (CRC <> Stored_CRC);
    
IF Changed THEN
    Stored_CRC := CRC;
END_IF
END_METHOD

END_FUNCTION_BLOCK

// Classes/Function Block Wrappers/Classes/T_ValueMonitor
{attribute 'no_explicit_call':= 'do not call this POU directly'}
FUNCTION_BLOCK T_ValueMonitor
VAR
    _CurrentValue : INT := -1;
    _PreviousValue : INT;
    _Changed : BOOL;
END_VAR

PROPERTY Changed : BOOL
GET
Changed := _Changed;
END_GET
END_PROPERTY

PROPERTY CurrentValue : INT
GET
CurrentValue := _CurrentValue;
END_GET
END_PROPERTY

PROPERTY PreviousValue : INT
GET
PreviousValue := _PreviousValue;
END_GET
END_PROPERTY

METHOD Reset
VAR_INPUT
END_VAR
_CurrentValue := 0;
_PreviousValue := 0;
END_METHOD

METHOD Test : BOOL
VAR_INPUT
    Value : INT;
END_VAR
_Changed := Value <> _CurrentValue;
_PreviousValue := _CurrentValue;
_CurrentValue := Value;

Test := _Changed;
END_METHOD

END_FUNCTION_BLOCK

// Classes/Function Block Wrappers/Classes/T_ValueMonitorEx
{attribute 'no_explicit_call':= 'do not call this POU directly'}
FUNCTION_BLOCK T_ValueMonitorEx
VAR
    _Changed : BOOL;
    StoredValue : ARRAY[0..7] OF BYTE;
END_VAR

PROPERTY Changed : BOOL
GET
Changed := _Changed;
END_GET
END_PROPERTY

METHOD Reset
VAR_INPUT
END_VAR
MEMSET(
    destAddr := ADR(StoredValue),
    fillByte  := 16#00,
    n        := SIZEOF(StoredValue));
END_METHOD

METHOD Test : BOOL;
VAR_INPUT
    Value : ANY_NUM;
END_VAR
_Changed := 0 <>  MEMCMP(
                    pBuf1 := Value.pValue,
                    pBuf2 := ADR(StoredValue),
                    n     := DINT_TO_UDINT(Value.diSize));
    
IF _Changed THEN
    MEMCPY(
        destAddr := ADR(StoredValue),
        srcAddr  := Value.pValue,
        n        := DINT_TO_UDINT(Value.diSize));
END_IF

Test := _Changed;
END_METHOD

END_FUNCTION_BLOCK

// Classes/Function Block Wrappers/Event Logging/F_LogError
FUNCTION F_LogError  
VAR_INPUT
    Source  : T_MaxString;
    Message : T_MaxString;
END_VAR

ADSLOGSTR(
        msgCtrlMask := ADSLOG_MSGTYPE_STRING OR ADSLOG_MSGTYPE_ERROR OR ADSLOG_MSGTYPE_LOG,
        msgFmtStr := F_FormatStringEx2('%s : %s',Source,Message),
        strArg := '');

END_FUNCTION

// Classes/Function Block Wrappers/Event Logging/F_LogMessage
FUNCTION F_LogMessage : T_MaxString
VAR_INPUT
    Source  : T_MaxString;
    Message : T_MaxString;
END_VAR

ADSLOGSTR(
    msgCtrlMask := ADSLOG_MSGTYPE_STRING OR ADSLOG_MSGTYPE_HINT OR ADSLOG_MSGTYPE_LOG,
    msgFmtStr := F_FormatStringEx2('%s : %s',Source,Message),
    strArg := '');

END_FUNCTION

// Classes/Function Block Wrappers/Event Logging/F_LogWarning
FUNCTION F_LogWarning : T_MaxString 
VAR_INPUT
    Source  : T_MaxString;
    Message : T_MaxString;
END_VAR

ADSLOGSTR(
    msgCtrlMask := ADSLOG_MSGTYPE_STRING OR ADSLOG_MSGTYPE_WARN OR ADSLOG_MSGTYPE_LOG,
    msgFmtStr := F_FormatStringEx2('%s : %s',Source,Message),
    strArg := '');

END_FUNCTION

// Classes/Notifications/Handler Interface/T_NotificationHandler
FUNCTION_BLOCK T_NotificationHandler IMPLEMENTS I_NotificationHandler
VAR
    _NotificationArgs : T_Stream(StreamLength := 4);
    _Raised : BOOL;
END_VAR

METHOD IsRaised : BOOL;
VAR_INPUT
END_VAR
IsRaised := _Raised;
_Raised := FALSE;
END_METHOD

PROPERTY NotificationArgs : I_StreamReader
GET
NotificationArgs := _NotificationArgs;
END_GET
END_PROPERTY

METHOD OnNotificationReceived
VAR_INPUT
	NotificationId	  : UDINT;
	NotificationName  : Tc2_System.T_MaxString;
	Args	          : I_StreamReader;
END_VAR
VAR
    i : UDINT;
    ByteToCopy : BYTE;
END_VAR
IF Args.ByteCount > 0 THEN // has event arguments..
    _NotificationArgs.CopyFromStreamReader(Args);
END_IF
_NotificationArgs.Seek(0);

_Raised := TRUE;
END_METHOD

END_FUNCTION_BLOCK

// Classes/Notifications/List Of Handlers/T_ListONotificationHandlers
{attribute 'hide'}
FUNCTION_BLOCK T_ListONotificationHandlers
VAR
    Buffer : FB_DynMem_Buffer(ipMemMan:= DynamicMemoryManager);
    DynamicMemoryManager : FB_DynMem_Manager;

    pHandler : POINTER TO I_NotificationHandler;
    HandlerCount : UDINT;
    Capacity : UDINT;
END_VAR

METHOD AddHandler
VAR_INPUT
    Handler : I_NotificationHandler;
END_VAR
IF Count = Capacity THEN
    Capacity := Capacity * 2;
    Buffer.Resize(
        nSize     := Capacity * SIZEOF(PVOID),
        bPreserve := TRUE,
        bReset    := FALSE);
    pHandler := Buffer.pBuffer;
END_IF

pHandler[HandlerCount] := Handler;
HandlerCount := HandlerCount + 1;
END_METHOD

METHOD Clear
VAR_INPUT
END_VAR
Buffer.Clear();
HandlerCount := 0;
END_METHOD

PROPERTY Count : UDINT
GET
Count := HandlerCount;
END_GET
END_PROPERTY

METHOD FB_exit : BOOL
VAR_INPUT
	bInCopyCode : BOOL; // if TRUE, the exit method is called for exiting an instance that is copied afterwards (online change).
END_VAR
IF NOT bInCopyCode THEN
    Buffer.DeleteBuffer();
    pHandler := 0;
END_IF
END_METHOD

METHOD FB_init : BOOL
VAR_INPUT
	bInitRetains : BOOL; // if TRUE, the retain variables are initialized (warm start / cold start)
	bInCopyCode : BOOL;  // if TRUE, the instance afterwards gets moved into the copy code (online change)
    Capacity : UDINT;
END_VAR
Buffer.CreateBuffer(
    nSize := Capacity * SIZEOF(PVOID),
    bReset := TRUE);
    
pHandler := Buffer.pBuffer;
THIS^.Capacity := Capacity;
END_METHOD

METHOD GetHandler : I_NotificationHandler
VAR_INPUT
    Index : UDINT;
END_VAR
IF Index < HandlerCount AND Index >= 0 THEN 
    GetHandler := pHandler[Index];
END_IF
END_METHOD

END_FUNCTION_BLOCK

// Classes/Notifications/Notification Class/T_Notification
{attribute 'reflection'}
FUNCTION_BLOCK T_Notification IMPLEMENTS I_Notification
VAR
    {attribute 'instance-path'} {attribute 'no_init'}
    FullName : T_MaxString; // Automatically initialised with the full name of the instance   
    
    EventHandlers : T_ListONotificationHandlers(Capacity := 5);
    
    _Name : T_MaxString; // stripped version
    _Args : T_Stream(StreamLength := 8);
    _NotificationId : UDINT := 999999; // initialise with unlikely notification id to catch cases where it is not initialised by client code
END_VAR

METHOD AddNotificationHandler : I_Notification
VAR_INPUT
    Handler : I_NotificationHandler;
END_VAR
EventHandlers.AddHandler(Handler);
AddNotificationHandler := THIS^;
END_METHOD

METHOD ClearNotificationHandlers : I_Notification
EventHandlers.Clear();
ClearNotificationHandlers := THIS^;
END_METHOD

METHOD FB_init : BOOL
VAR_INPUT
	bInitRetains : BOOL; // if TRUE, the retain variables are initialized (warm start / cold start)
	bInCopyCode : BOOL;  // if TRUE, the instance afterwards gets moved into the copy code (online change)
END_VAR
VAR
    
END_VAR
THIS^._Name := stripName(FullName);
END_METHOD

METHOD Raise
VAR
    Handler : I_NotificationHandler;
    i : UDINT;
END_VAR
IF EventHandlers.Count > 0 THEN
    FOR i := 0 TO EventHandlers.Count - 1 DO
        Handler := EventHandlers.GetHandler(i);
        IF Handler <> 0 THEN
            _Args.Seek(0); // to ensure that each handler reads args from start of the stream
            Handler.OnNotificationReceived(
                NotificationId   := _NotificationId,
                NotificationName := _Name,
                Args             := _Args);
        END_IF
    END_FOR
END_IF
_Args.Clear(); // to leave event args empty for next time event is raised
END_METHOD

METHOD SetNotificationId : I_Notification
VAR_INPUT
    NotificationId : UDINT;
END_VAR
_NotificationId   := NotificationId;
SetNotificationId := THIS^;
END_METHOD

METHOD PRIVATE stripName : T_MaxString
VAR_INPUT
    FullName : T_MaxString;
END_VAR
VAR
    StringSplitter : T_StringSplitter;
    Result : T_MaxString;
END_VAR
StringSplitter.Init(
    Str := FullName,
    Delim1 := '.',
    Delim2 := '');
    
WHILE StringSplitter.HasMore() DO
    Result := StringSplitter.GetNext(); // to get last sub-section
END_WHILE

StripName := Result;
END_METHOD

PROPERTY PUBLIC Args : I_StreamWriter
GET
Args := _Args;
END_GET
END_PROPERTY

PROPERTY Name : T_MaxString
GET
Name := _Name;
END_GET
END_PROPERTY

PROPERTY NotificationId : UDINT
GET
NotificationId := _NotificationId;
END_GET
SET
_NotificationId := NotificationId;
END_SET
END_PROPERTY

END_FUNCTION_BLOCK

// Events/Assertion Failed/I_EventHandler_OnAssertionFailed
INTERFACE I_EventHandler_OnAssertionFailed EXTENDS I_EventHandlerBase

METHOD OnAssertionFailed
VAR_INPUT
    EventArgs   : I_StreamReader;
END_VAR
END_METHOD

END_INTERFACE

// Events/Assertion Failed/T_Event_AssertionFailed
FUNCTION_BLOCK T_Event_AssertionFailed EXTENDS T_EventBase IMPLEMENTS I_Event
VAR
    Message : T_MaxString;
    Handler : I_EventHandler_OnAssertionFailed;
END_VAR

METHOD  CallHandler
VAR_INPUT
    HandlerBase : I_EventHandlerBase;
    EventArgs   : I_StreamReader;
END_VAR
IF __QUERYINTERFACE(HandlerBase,Handler) THEN
    Message := EventArgs.Read_STRING();
    Handler.OnAssertionFailed(EventArgs);
END_IF
END_METHOD

METHOD  IsHandlerSupported : BOOL
VAR_INPUT
    HandlerBase : I_EventHandlerBase;
END_VAR
IF __QUERYINTERFACE(HandlerBase,Handler) THEN
    IsHandlerSupported := TRUE;
END_IF
END_METHOD

END_FUNCTION_BLOCK

// Events/Execution Aborted/I_EventHandler_OnExecutionAborted
INTERFACE I_EventHandler_OnExecutionAborted EXTENDS I_EventHandlerBase

METHOD OnExecutionAborted
VAR_INPUT
    Message : T_MaxString;
END_VAR
END_METHOD

END_INTERFACE

// Events/Execution Aborted/T_Event_ExecutionAborted
FUNCTION_BLOCK T_Event_ExecutionAborted EXTENDS T_EventBase IMPLEMENTS I_Event
VAR
    Message : T_MaxString;
    Handler : I_EventHandler_OnExecutionAborted;
END_VAR

METHOD  CallHandler
VAR_INPUT
    HandlerBase : I_EventHandlerBase;
    EventArgs   : I_StreamReader;
END_VAR
VAR
    Message : T_MaxString;
END_VAR
IF __QUERYINTERFACE(HandlerBase,Handler) THEN
    Message := EventArgs.Read_STRING();
    Handler.OnExecutionAborted(Message);
END_IF
END_METHOD

METHOD  IsHandlerSupported : BOOL
VAR_INPUT
    HandlerBase : I_EventHandlerBase;
END_VAR
IF __QUERYINTERFACE(HandlerBase,Handler) THEN
    IsHandlerSupported := TRUE;
END_IF
END_METHOD

END_FUNCTION_BLOCK

// Events/Execution Failed/I_EventHandler_OnExecutionFailed
INTERFACE I_EventHandler_OnExecutionFailed EXTENDS I_EventHandlerBase

METHOD OnExecutionFailed
VAR_INPUT
    Message : T_MaxString;
END_VAR
END_METHOD

END_INTERFACE

// Events/Execution Failed/T_Event_ExecutionFailed
FUNCTION_BLOCK T_Event_ExecutionFailed EXTENDS T_EventBase IMPLEMENTS I_Event
VAR
    Message : T_MaxString;
    Handler : I_EventHandler_OnExecutionFailed;
END_VAR

METHOD  CallHandler
VAR_INPUT
    HandlerBase : I_EventHandlerBase;
    EventArgs   : I_StreamReader;
END_VAR
VAR
    Message : T_MaxString;
END_VAR
IF __QUERYINTERFACE(HandlerBase,Handler) THEN
    Message := EventArgs.Read_STRING();
    Handler.OnExecutionFailed(Message);
END_IF
END_METHOD

METHOD  IsHandlerSupported : BOOL
VAR_INPUT
    HandlerBase : I_EventHandlerBase;
END_VAR
IF __QUERYINTERFACE(HandlerBase,Handler) THEN
    IsHandlerSupported := TRUE;
END_IF
END_METHOD

END_FUNCTION_BLOCK

// Functions/F_Assert
FUNCTION F_Assert : BOOL
VAR_INPUT
    Assertion : BOOL;
    FailMessage : T_MaxString;
END_VAR
VAR_STAT
    AssertionMessage : FB_TcMessage;
    AssertionSourceInfo : FB_TcSourceInfo;
END_VAR

F_Assert := Assertion;
IF Assertion = FALSE THEN
    // Send assertion message to Event Logger...
//    IF NOT AssertionMessage.EqualsToEventClass(TC_EVENTS.tcl_BaseClassEvents.AssertionFailed.uuidEventClass) THEN
//        AssertionSourceInfo.sName := 'F_Assert';
//        AssertionMessage.CreateEx(
//            stEventEntry := TC_EVENTS.tcl_BaseClassEvents.AssertionFailed,
//            ipSourceInfo := AssertionSourceInfo);
//    END_IF
//    AssertionMessage.ipArguments.Clear().AddStringByValue(FailMessage);
//    AssertionMessage.Send(0);
    
    GlobalEvents.Event_AssertionFailed.Args
        .Clear()
        .Add_STRING(FailMessage);
    GlobalEvents.Event_AssertionFailed.Raise(); // to allow the machine to abort on any assertion failure
    
    GlobalEvents.Notification_AssertionFailed.Args
        .Clear()
        .Add_STRING(FailMessage);
    GlobalEvents.Notification_AssertionFailed.Raise(); // to allow the machine to abort on any assertion failure
    
END_IF

END_FUNCTION

// Functions/F_ClearMem
FUNCTION F_ClearMem : BOOL
VAR_INPUT
    Data : ANY;
END_VAR
VAR
END_VAR

MEMSET(
    destAddr := Data.pValue,
    fillByte := 0,
    n        := DINT_TO_UDINT(Data.diSize));

END_FUNCTION

// Functions/F_DINT_TO_UDINT
FUNCTION F_DINT_TO_UDINT : UDINT
VAR_INPUT
    value : DINT;
END_VAR
VAR
    inRangeValue : DINT;
END_VAR

F_Assert(
    Assertion := value >= 0,
    FailMessage := 'Input arg of F_DINT_TO_UDINT was < 0 so value of 0 was returned');

inRangeValue := MAX(0,value);
F_DINT_TO_UDINT := DINT_TO_UDINT(inRangeValue);

END_FUNCTION

// Functions/F_Equals
FUNCTION F_Equals : BOOL
VAR_INPUT
    In1 : LREAL;
    In2 : LREAL;
    Delta : LREAL;
END_VAR
VAR
    Difference : LREAL;
END_VAR

Difference := ABS(In1 - In2);
F_Equals := Difference < Delta;

END_FUNCTION

// Functions/F_GetAdsPort
FUNCTION F_GetAdsPort : UINT
VAR
    TaskIndex : DINT;
END_VAR

TaskIndex := GETCURTASKINDEXEX();
IF TaskIndex > 0 THEN
    F_GetAdsPort := TwinCAT_SystemInfoVarList._AppInfo.AdsPort;
END_IF

END_FUNCTION

// Functions/F_GetTaskTime
FUNCTION F_GetTaskTime : LREAL
VAR
	TaskIndex: DINT;
END_VAR

TaskIndex := GETCURTASKINDEXEX();
IF TaskIndex > 0 THEN
    F_GetTaskTime := UDINT_TO_LREAL(TwinCAT_SystemInfoVarList._taskInfo[TaskIndex].CycleTime) * LREAL#1E-7;
END_IF

END_FUNCTION

// Functions/F_NotEqual
FUNCTION F_NotEqual : BOOL
VAR_INPUT
    In1 : LREAL;
    In2 : LREAL;
    Delta : LREAL;
END_VAR
VAR
    Difference : LREAL;
END_VAR

Difference := ABS(In1 - In2);
F_NotEqual := Difference > Delta;

END_FUNCTION

// Functions/F_UDINT_TO_DINT
FUNCTION F_UDINT_TO_DINT : DINT
VAR_INPUT
    value : UDINT;
END_VAR
VAR
    inRangeValue : UDINT;
END_VAR

IF value.31 THEN // out of range
    F_Assert(
        Assertion := FALSE,
        FailMessage := 'Input arg of F_UDINT_TO_DINT too large to convert, so value of Max DINT (2147483647) was returned');

    inRangeValue := 16#7FFF_FFFF; // ‭Max DINT = 2147483647‬
ELSE
    inRangeValue := value;
END_IF
F_UDINT_TO_DINT := UDINT_TO_DINT(inRangeValue);

END_FUNCTION
